INTERFACE ITF_Tool_1

METHOD Grip : BOOL
VAR_INPUT
END_VAR
END_METHOD

METHOD Release : BOOL
VAR_INPUT
END_VAR
END_METHOD

END_INTERFACE

(* stored: Version 1.1.0.1, ProductVersion 3.1.4026.18
   Itf ITF_Tool_1: Id {8875c691-5b54-47cc-8d93-e74cb61af3bb}
   Method Grip: Id {b0f27820-f07d-4f08-ae06-84bac441a464}
   Method Release: Id {03a3e0db-4772-4093-ac28-d41cdb549f9b} *)
